(* CODESYS project bl20_medianFilterForStable.project

Project tree, tasks and I/O mapping:
  Device : BL20-PG-EN-V3, Turck, order no. 6827393, version 3.5.11.20
    application Application
      libraries: BLxxFB Local IO, 1.1.1.0 (TURCK); BASIC, 3.31 (OSCAT); Util, * (System); VisuDialogs, * (System)
      task MainTask (cyclic, interval t#20ms, priority 1) calls PLC_PRG
      task TrendRecordingTask (cyclic, interval 100 ms, priority 31) calls VisuTrendStorageAccess.GlobalInstances.g_TrendRecordingManager.CyclicCall
      program PLC_PRG [ST]
      visualisation Visualization
      function FC_InsertionSortAndFilter [ST]
      Trend Recording Manager
        Visualization_Trend1
    Gateway_LED_APPL : Gateway LED APPL, Turck, version 1.0.3.0
        unmapped channels: Applikation LED (Grün), Applikation LED (Rot), Reserved, Reserved, Reserved, Reserved, Reserved, Reserved
    Local_IO_BL20 : Local IO BL20, Turck, version 1.1.3.0
      BL20_4AI_U_I : BL20-4AI-U/I, Turck, version 1.1.3.0
          input  Application.PLC_PRG.wRawInput : WORD  // Input value Ch1
          unmapped channels: Input value Ch2, Input value Ch3, Input value Ch4, Measured value out of range Ch1, Wire break  Ch1, Over--underflow Ch1, Measured value out of range Ch2, Wire break  Ch2, Over--underflow Ch2, Measured value out of range Ch3, Wire break  Ch3, Over--underflow Ch3, Measured value out of range Ch4, Wire break  Ch4, Over--underflow Ch4, Dummy, Dummy, Dummy, Dummy
      BL20_E_8DI_24VDC_P : BL20-E-8DI-24VDC-P, Turck, version 1.1.3.0
          unmapped channels: Input value Ch1, Input value Ch2, Input value Ch3, Input value Ch4, Input value Ch5, Input value Ch6, Input value Ch7, Input value Ch8
  text list GlobalTextList
*)

// Device/Application/PLC_PRG
PROGRAM PLC_PRG
VAR CONSTANT
	iArraySize : INT := 99;
END_VAR

VAR
	awInput : ARRAY[0..iArraySize] OF WORD;	
	wRawInput : WORD;
	diResult : DINT;
	i,j : INT;
	
	rRawDistance : REAL;
	rFilterDistance : REAL;
	
	rScale: REAL := 1;
	rOffset: REAL := 0;
END_VAR


IF i < iArraySize THEN
	awInput[i] := wRawInput;
	i := i + 1;
ELSE

	FOR j := 0 TO iArraySize DO
		IF j < iArraySize -1 THEN
			awInput[j] := awInput[j+1];			
		ELSE
			awInput[j] := wRawInput;			
		END_IF
	END_FOR 
	diResult := FC_InsertionSortAndFilter(awInput:= awInput);
	//i := 0;
END_IF

rRawDistance := WORD_TO_REAL(wRawInput) * rScale + rOffset;
rFilterDistance := DINT_TO_REAL(diResult) * rScale + rOffset;

END_PROGRAM

// Device/Application/FC_InsertionSortAndFilter
FUNCTION FC_InsertionSortAndFilter : DINT;
VAR_IN_OUT
	awInput : ARRAY[*] OF WORD;	
END_VAR

VAR_INPUT
END_VAR
VAR
	diLB : DINT;
	diUB : DINT;
	i, j : DINT;
	wKey : WORD;
	
	diMinIndex : DINT;
	diMaxIndex : DINT;	
	diInterval : DINT;
	
	diDividerFactor: DINT := 10;
	
	k : DINT;
	filteredSum : UDINT;
END_VAR

//입력 ARRAY 시작 및 끝 확인 
diLB:= LOWER_BOUND(awInput, 1);
diUB:= UPPER_BOUND(awInput, 1);

// Insertion Sort 수행
FOR i:=diLB TO diUB BY 1 DO
	wKey := awInput[i];
	
	FOR j:= i-1 TO 0 BY -1 DO
		IF awInput[j] > wKey THEN
			awInput[j+1] := awInput[j];
		ELSE
			EXIT; 
		END_IF
	END_FOR
	awInput[j+1] := wKey; 
END_FOR

// Median Filter 적용 25~75%용 구간 설정
diInterval := (diUB-diLB)/4;
diMinIndex := diLB + diInterval;
diMaxIndex := diUB - diInterval;

FOR k:= diMinIndex TO diMaxIndex DO
	filteredSum := filteredSum + awInput[k] ;
END_FOR

// Median Filter 적용된 내용만 평균 계산 후 리턴
FC_InsertionSortAndFilter := UDINT_TO_DINT(filteredSum / DINT_TO_UDINT(diMaxIndex-diMinIndex+1));

END_FUNCTION

// Device/Application/Visualization
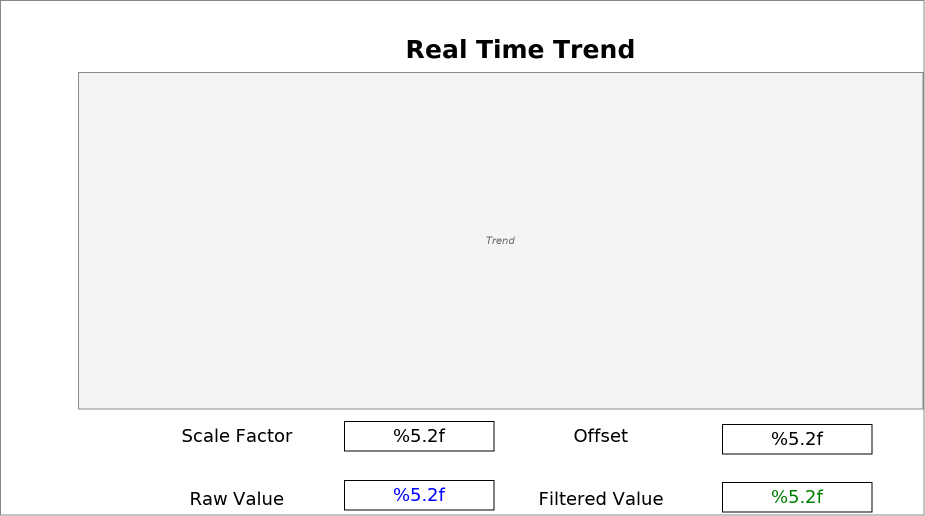
VISUALIZATION Visualization  // 925x516
    Trend (78,72 845x337)
        p2423372160: tt h:mm:ss
        p2833066001: Visualization_Trend1
    Label (322,34 397x30), "Real Time Trend"
    RoundedRectangle (344,421 150x30), "%5.2f", text variable: PLC_PRG.rScale
        OnMouseClick: write the text variable via Default
    Label (162,421 150x30), "Scale Factor"
    Label (526,421 150x30), "Offset"
    Label (162,484 150x30), "Raw Value"
    Label (526,484 150x30), "Filtered Value"
    RoundedRectangle (722,424 150x30), "%5.2f", text variable: PLC_PRG.rOffset
        OnMouseClick: write the text variable via Default
    RoundedRectangle (344,480 150x30), "%5.2f", text variable: PLC_PRG.rRawDistance
    RoundedRectangle (722,482 150x30), "%5.2f", text variable: PLC_PRG.rFilterDistance
END_VISUALIZATION
